{attribute addProperty BoxType "EM7004-0000-0017"}
{attribute addProperty Id "ControlAT %Q*Control_84750349162"}
{attribute addProperty CRC "3640114352"}
{attribute addProperty SizeInBites "16"}
{attribute addProperty SizeInBytes "2"}
TYPE PLS_Outputs_D8F7BCB0 :
STRUCT
	{attribute addProperty Name "Control"}
	Control AT %Q* : Control_84750349;
END_STRUCT
END_TYPE

(* stored: Version 1.2.0.0, ProductVersion 3.1.4024.9
   DUT PLS_Outputs_D8F7BCB0: Id {78119381-f63b-44b8-93dd-343a3f89d19d} *)
